// TIA Portal V20 export
FUNCTION "OneMES_HMI_Control" : Void   // FC20230, LAD
{ S7_Optimized_Access := 'TRUE' }
// stored: AutoNumber false, SetENOAutomatically false
   VAR_INPUT
      iManualMode : Bool;
      iOP_Sum : SInt;
   END_VAR
   VAR_IN_OUT
      ioHMI : "UDT_OneMES_HMI_Control";
      ioOP : Array[1.."OP_Sum"] of "UDT_MESControl";
      ioPluse : Bool;
   END_VAR
   VAR_TEMP   // added for the SCL form of the ladder/FBD networks
      _w1 : Bool;
   END_VAR
BEGIN

REGION Network 1: OP Limit
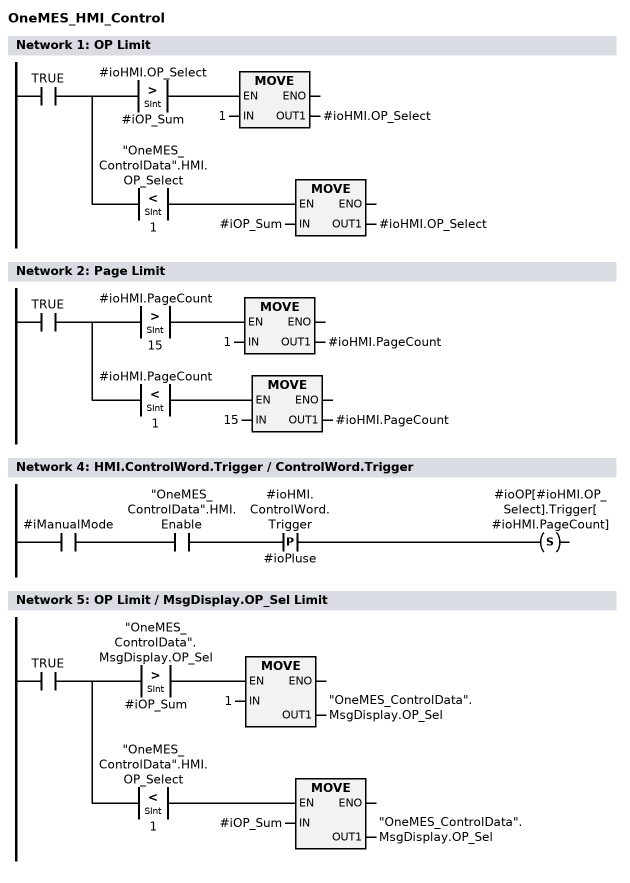
   RUNG wire#powerrail
      Contact( TRUE )
      wire#w1
      { S7_Templates := "SrcType := SInt" } GT_Contact(in1 := #ioHMI.OP_Select, in2 := #iOP_Sum)
      Move(in := 1, out1 => #ioHMI.OP_Select)
   END_RUNG
   RUNG wire#w1
      { S7_Templates := "SrcType := SInt" } LT_Contact(in1 := "OneMES_ControlData".HMI.OP_Select, in2 := 1)
      Move(in := #iOP_Sum, out1 => #ioHMI.OP_Select)
   END_RUNG
   // the same network as SCL:
   IF TRUE AND (#ioHMI.OP_Select > #iOP_Sum) THEN #ioHMI.OP_Select := 1; END_IF;
   IF TRUE AND ("OneMES_ControlData".HMI.OP_Select < 1) THEN #ioHMI.OP_Select := #iOP_Sum; END_IF;
END_REGION

REGION Network 2: Page Limit
   RUNG wire#powerrail
      Contact( TRUE )
      wire#w1
      { S7_Templates := "SrcType := SInt" } GT_Contact(in1 := #ioHMI.PageCount, in2 := 15)
      Move(in := 1, out1 => #ioHMI.PageCount)
   END_RUNG
   RUNG wire#w1
      { S7_Templates := "SrcType := SInt" } LT_Contact(in1 := #ioHMI.PageCount, in2 := 1)
      Move(in := 15, out1 => #ioHMI.PageCount)
   END_RUNG
   // the same network as SCL:
   IF TRUE AND (#ioHMI.PageCount > 15) THEN #ioHMI.PageCount := 1; END_IF;
   IF TRUE AND (#ioHMI.PageCount < 1) THEN #ioHMI.PageCount := 15; END_IF;
END_REGION

REGION Network 3 (SCL): Copy HMI Data
   #ioHMI.ControlWord.StepNO := #ioOP[#ioHMI.OP_Select].StepNO[#ioHMI.PageCount];
   #ioHMI.ControlWord.FaultCode := #ioOP[#ioHMI.OP_Select].FaultCode[#ioHMI.PageCount];
   #ioHMI.ControlWord.Busy := #ioOP[#ioHMI.OP_Select].Busy[#ioHMI.PageCount];
   #ioHMI.ControlWord.ResultOK := #ioOP[#ioHMI.OP_Select].ResultOK[#ioHMI.PageCount];
   #ioHMI.ControlWord.ResultNG := #ioOP[#ioHMI.OP_Select].ResultNG[#ioHMI.PageCount];
   IF NOT #iManualMode THEN
       #ioHMI.Enable := 0;
   END_IF;
END_REGION

REGION Network 4: HMI.ControlWord.Trigger / ControlWord.Trigger
   RUNG wire#powerrail
      Contact( #iManualMode )
      Contact( "OneMES_ControlData".HMI.Enable )
      P_Contact(operand := #ioHMI.ControlWord.Trigger, bit := #ioPluse)
      S_Coil( #ioOP[#ioHMI.OP_Select].Trigger[#ioHMI.PageCount] )
   END_RUNG
   // the same network as SCL:
   #_w1 := #iManualMode AND "OneMES_ControlData".HMI.Enable AND #ioHMI.ControlWord.Trigger AND NOT #ioPluse;   // rising edge of #ioHMI.ControlWord.Trigger
   #ioPluse := #ioHMI.ControlWord.Trigger;
   IF #_w1 THEN #ioOP[#ioHMI.OP_Select].Trigger[#ioHMI.PageCount] := TRUE; END_IF;
END_REGION

REGION Network 5: OP Limit / MsgDisplay.OP_Sel Limit
   RUNG wire#powerrail
      Contact( TRUE )
      wire#w1
      { S7_Templates := "SrcType := SInt" } GT_Contact(in1 := "OneMES_ControlData".MsgDisplay.OP_Sel, in2 := #iOP_Sum)
      Move(in := 1, out1 => "OneMES_ControlData".MsgDisplay.OP_Sel)
   END_RUNG
   RUNG wire#w1
      { S7_Templates := "SrcType := SInt" } LT_Contact(in1 := "OneMES_ControlData".HMI.OP_Select, in2 := 1)
      Move(in := #iOP_Sum, out1 => "OneMES_ControlData".MsgDisplay.OP_Sel)
   END_RUNG
   // the same network as SCL:
   IF TRUE AND ("OneMES_ControlData".MsgDisplay.OP_Sel > #iOP_Sum) THEN
       "OneMES_ControlData".MsgDisplay.OP_Sel := 1;
   END_IF;
   IF TRUE AND ("OneMES_ControlData".HMI.OP_Select < 1) THEN
       "OneMES_ControlData".MsgDisplay.OP_Sel := #iOP_Sum;
   END_IF;
END_REGION

REGION Network 6 (SCL)
   CASE "OneMES_ControlData".HMI.OP_Select OF
       1:
           "OneMES_ControlData".MsgDisplay.DB_NO1 := 2001;
           "OneMES_ControlData".MsgDisplay.DB_NO2 := 2002;
           "OneMES_ControlData".MsgDisplay.DB_NO3 := 2003;
           "OneMES_ControlData".MsgDisplay.DB_NO4 := 2004;
           "OneMES_ControlData".MsgDisplay.DB_NO5 := 2005;
           "OneMES_ControlData".MsgDisplay.DB_NO6 := 2006;
           "OneMES_ControlData".MsgDisplay.DB_NO7 := 2007;

       2:
           "OneMES_ControlData".MsgDisplay.DB_NO1 := 2011;
           "OneMES_ControlData".MsgDisplay.DB_NO2 := 2012;
           "OneMES_ControlData".MsgDisplay.DB_NO3 := 2013;
           "OneMES_ControlData".MsgDisplay.DB_NO4 := 2014;
           "OneMES_ControlData".MsgDisplay.DB_NO5 := 2015;
           "OneMES_ControlData".MsgDisplay.DB_NO6 := 2016;
           "OneMES_ControlData".MsgDisplay.DB_NO7 := 2017;

       3:
           "OneMES_ControlData".MsgDisplay.DB_NO1 := 2021;
           "OneMES_ControlData".MsgDisplay.DB_NO2 := 2022;
           "OneMES_ControlData".MsgDisplay.DB_NO3 := 2023;
           "OneMES_ControlData".MsgDisplay.DB_NO4 := 2024;
           "OneMES_ControlData".MsgDisplay.DB_NO5 := 2025;
           "OneMES_ControlData".MsgDisplay.DB_NO6 := 2026;
           "OneMES_ControlData".MsgDisplay.DB_NO7 := 2027;

       4:
           "OneMES_ControlData".MsgDisplay.DB_NO1 := 2031;
           "OneMES_ControlData".MsgDisplay.DB_NO2 := 2032;
           "OneMES_ControlData".MsgDisplay.DB_NO3 := 2033;
           "OneMES_ControlData".MsgDisplay.DB_NO4 := 2034;
           "OneMES_ControlData".MsgDisplay.DB_NO5 := 2035;
           "OneMES_ControlData".MsgDisplay.DB_NO6 := 2036;
           "OneMES_ControlData".MsgDisplay.DB_NO7 := 2037;

       5:
           "OneMES_ControlData".MsgDisplay.DB_NO1 := 2041;
           "OneMES_ControlData".MsgDisplay.DB_NO2 := 2042;
           "OneMES_ControlData".MsgDisplay.DB_NO3 := 2043;
           "OneMES_ControlData".MsgDisplay.DB_NO4 := 2044;
           "OneMES_ControlData".MsgDisplay.DB_NO5 := 2045;
           "OneMES_ControlData".MsgDisplay.DB_NO6 := 2046;
           "OneMES_ControlData".MsgDisplay.DB_NO7 := 2047;

       // ELSE  "OneMES_ControlData".MsgDisplay.OP_Sel :=1
       //     ;
   END_CASE;
END_REGION

REGION Network 7 (SCL): MES Msg Display
   CASE "OneMES_ControlData".HMI.OP_Select OF
       1:
           "OneMES_ControlData".MsgDisplay.PLC_RequestTimeOutCount_Offset := 6; 
          "OneMES_ControlData".MsgDisplay.PLC_RequestTransaction_ID_Offset := 8;
          "OneMES_ControlData".MsgDisplay.PLC_RequestSignal_Offset := 12;
          "OneMES_ControlData".MsgDisplay.MES_ResponseError_ID_Offset := 14;
          "OneMES_ControlData".MsgDisplay.MES_ResponseSignal_Offset := 16;

      2:
          "OneMES_ControlData".MsgDisplay.PLC_RequestTimeOutCount_Offset := 18;
          "OneMES_ControlData".MsgDisplay.PLC_RequestTransaction_ID_Offset := 8;
          "OneMES_ControlData".MsgDisplay.PLC_RequestSignal_Offset := 20;
          "OneMES_ControlData".MsgDisplay.MES_ResponseError_ID_Offset := 22;
          "OneMES_ControlData".MsgDisplay.MES_ResponseSignal_Offset := 24;

      3:
          "OneMES_ControlData".MsgDisplay.PLC_RequestTimeOutCount_Offset := 26;
          "OneMES_ControlData".MsgDisplay.PLC_RequestTransaction_ID_Offset := 28;
          "OneMES_ControlData".MsgDisplay.PLC_RequestSignal_Offset := 32;
          "OneMES_ControlData".MsgDisplay.MES_ResponseError_ID_Offset := 34;
          "OneMES_ControlData".MsgDisplay.MES_ResponseSignal_Offset := 36;

      4:
          "OneMES_ControlData".MsgDisplay.PLC_RequestTimeOutCount_Offset := 38;
          "OneMES_ControlData".MsgDisplay.PLC_RequestTransaction_ID_Offset := 40;
          "OneMES_ControlData".MsgDisplay.PLC_RequestSignal_Offset := 44;
          "OneMES_ControlData".MsgDisplay.MES_ResponseError_ID_Offset := 46;
          "OneMES_ControlData".MsgDisplay.MES_ResponseSignal_Offset := 48;

      5:
          "OneMES_ControlData".MsgDisplay.PLC_RequestTimeOutCount_Offset := 50;
          "OneMES_ControlData".MsgDisplay.PLC_RequestTransaction_ID_Offset := 52;
          "OneMES_ControlData".MsgDisplay.PLC_RequestSignal_Offset := 56;
          "OneMES_ControlData".MsgDisplay.MES_ResponseError_ID_Offset := 58;
          "OneMES_ControlData".MsgDisplay.MES_ResponseSignal_Offset := 60;

      6:
          "OneMES_ControlData".MsgDisplay.PLC_RequestTimeOutCount_Offset := 62;
          "OneMES_ControlData".MsgDisplay.PLC_RequestTransaction_ID_Offset := 64;
          "OneMES_ControlData".MsgDisplay.PLC_RequestSignal_Offset := 68;
          "OneMES_ControlData".MsgDisplay.MES_ResponseError_ID_Offset := 70;
          "OneMES_ControlData".MsgDisplay.MES_ResponseSignal_Offset := 72;

      7:
          "OneMES_ControlData".MsgDisplay.PLC_RequestTimeOutCount_Offset := 74;
          "OneMES_ControlData".MsgDisplay.PLC_RequestTransaction_ID_Offset := 76;
          "OneMES_ControlData".MsgDisplay.PLC_RequestSignal_Offset := 80;
          "OneMES_ControlData".MsgDisplay.MES_ResponseError_ID_Offset := 82;
          "OneMES_ControlData".MsgDisplay.MES_ResponseSignal_Offset := 84;

      8:
          "OneMES_ControlData".MsgDisplay.PLC_RequestTimeOutCount_Offset := 86;
          "OneMES_ControlData".MsgDisplay.PLC_RequestTransaction_ID_Offset := 88;
          "OneMES_ControlData".MsgDisplay.PLC_RequestSignal_Offset := 92;
          "OneMES_ControlData".MsgDisplay.MES_ResponseError_ID_Offset := 94;
          "OneMES_ControlData".MsgDisplay.MES_ResponseSignal_Offset := 96;

      9:
          "OneMES_ControlData".MsgDisplay.PLC_RequestTimeOutCount_Offset := 98;
          "OneMES_ControlData".MsgDisplay.PLC_RequestTransaction_ID_Offset := 100;
          "OneMES_ControlData".MsgDisplay.PLC_RequestSignal_Offset := 104;
          "OneMES_ControlData".MsgDisplay.MES_ResponseError_ID_Offset := 106;
          "OneMES_ControlData".MsgDisplay.MES_ResponseSignal_Offset := 96;

      10:
          "OneMES_ControlData".MsgDisplay.PLC_RequestTimeOutCount_Offset := 108;
          "OneMES_ControlData".MsgDisplay.PLC_RequestTransaction_ID_Offset := 110;
          "OneMES_ControlData".MsgDisplay.PLC_RequestSignal_Offset := 114;
          "OneMES_ControlData".MsgDisplay.MES_ResponseError_ID_Offset := 116;
          "OneMES_ControlData".MsgDisplay.MES_ResponseSignal_Offset := 118;

      11:
          "OneMES_ControlData".MsgDisplay.PLC_RequestTimeOutCount_Offset := 120;
          "OneMES_ControlData".MsgDisplay.PLC_RequestTransaction_ID_Offset := 122;
          "OneMES_ControlData".MsgDisplay.PLC_RequestSignal_Offset := 126;
          "OneMES_ControlData".MsgDisplay.MES_ResponseError_ID_Offset := 128;
          "OneMES_ControlData".MsgDisplay.MES_ResponseSignal_Offset := 130;

      12:
          "OneMES_ControlData".MsgDisplay.PLC_RequestTimeOutCount_Offset := 132;
          "OneMES_ControlData".MsgDisplay.PLC_RequestTransaction_ID_Offset := 134;
          "OneMES_ControlData".MsgDisplay.PLC_RequestSignal_Offset := 138;
          "OneMES_ControlData".MsgDisplay.MES_ResponseError_ID_Offset := 140;
          "OneMES_ControlData".MsgDisplay.MES_ResponseSignal_Offset := 142;

      13:
          "OneMES_ControlData".MsgDisplay.PLC_RequestTimeOutCount_Offset := 152;
          "OneMES_ControlData".MsgDisplay.PLC_RequestTransaction_ID_Offset := 154;
          "OneMES_ControlData".MsgDisplay.PLC_RequestSignal_Offset := 158;
          "OneMES_ControlData".MsgDisplay.MES_ResponseError_ID_Offset := 160;
          "OneMES_ControlData".MsgDisplay.MES_ResponseSignal_Offset := 162;

      14:
          "OneMES_ControlData".MsgDisplay.PLC_RequestTimeOutCount_Offset := 170;
          "OneMES_ControlData".MsgDisplay.PLC_RequestTransaction_ID_Offset := 172;
          "OneMES_ControlData".MsgDisplay.PLC_RequestSignal_Offset := 176;
          "OneMES_ControlData".MsgDisplay.MES_ResponseError_ID_Offset := 178;
          "OneMES_ControlData".MsgDisplay.MES_ResponseSignal_Offset := 180;

      15:
          "OneMES_ControlData".MsgDisplay.PLC_RequestTimeOutCount_Offset := 6;
          "OneMES_ControlData".MsgDisplay.PLC_RequestTransaction_ID_Offset := 8;
          "OneMES_ControlData".MsgDisplay.PLC_RequestSignal_Offset := 12;
          "OneMES_ControlData".MsgDisplay.MES_ResponseError_ID_Offset := 14;
          "OneMES_ControlData".MsgDisplay.MES_ResponseSignal_Offset := 16;

       // ELSE  
       //     "OneMES_ControlData".MsgDisplay.Process_Sel:=1   ;
   END_CASE;
END_REGION
END_FUNCTION
